FUNCTION_BLOCK FB_LICTest EXTENDS FB_TestSuite
VAR
    (* Caller-owned axis, persistent storage, and Y motor.
       In a real PRG the AxisRef would come from MAIN.Mxx. *)
    axRef    : AXIS_REF;
    fbPDS    : LCLS_Tc_DevAbs.FB_PersistentDataStorage;

    (* FB_LIC is single-axis (nActiveMotorCount := 1), so only slot 1
       holds a real motor. aiMotionStage is sized to
       MotionConstants.MAX_STATE_MOTORS to match FB_LIC.FB_Init's
       fixed-size signature; slots 2-4 default-init to a nil interface
       and are never touched. *)
    fbMotorY : FB_MotionStageNC(AxisRef := axRef, iPersistentDataStorage := fbPDS, sName := 'Y');
    aiMotionStage : ARRAY[1..MotionConstants.MAX_STATE_MOTORS] OF I_MotionStage := [fbMotorY];

    {attribute 'pytmc' := '
        pv: MMS
        astPositionState.array: 1..4
    '}
    astPositionState : ARRAY[1..MotionConstants.MAX_STATE_MOTORS]
                         OF ARRAY[1..GeneralConstants.MAX_STATES] OF ST_PositionState;

    fbFFHWO    : FB_HardwareFFOutput;
    fbArbiter  : FB_Arbiter(1);
    fbSubSysIO : FB_DummyArbIO;

    (* Per-cycle caller-owned BOOL flags passed by reference to FB_LIC. *)
    bEnableMotion         : BOOL;
    bEnableBeamParams     : BOOL;
    bEnablePositionLimits : BOOL;
    bReadDBNow            : BOOL;

    (* Device-name strings bound to FB_LIC as REFERENCE TO STRING --
       a literal cannot be REF-bound, so they live as locals here. *)
    sDeviceName    : STRING := 'TST:LIC';
    sTransitionKey : STRING := 'TST:LIC-TRANSITION';

    fbLIC : FB_LIC(
        aiMotionStage         := aiMotionStage,
        astPositionState      := astPositionState,
        fbFFHWO               := fbFFHWO,
        fbArbiter             := fbArbiter,
        sDeviceName           := sDeviceName,
        sTransitionKey        := sTransitionKey,
        bEnableMotion         := bEnableMotion,
        bEnableBeamParams     := bEnableBeamParams,
        bEnablePositionLimits := bEnablePositionLimits,
        bReadDBNow            := bReadDBNow
    );

    (* Per-install PMPS-side state config (caller-owned). Mirrors what
       a real PRG_xxL0_LIC would declare. stDefault is the caller-owned
       baseline template that FB_CC_StatePMPSConfig's inner FB_StateSetup
       preloads from; fbLIC subsequently overrides per-state sName and
       fDelta via its own FB_CC_DeviceStateDefaults array. *)
    stDefault : ST_PositionState := (
        bMoveOk       := TRUE,
        bValid        := TRUE,
        bUseRawCounts := FALSE
    );

    afbStatePMPS : ARRAY[1..4] OF FB_CC_StatePMPSConfig[
        (stPositionState := astPositionState[1][E_LIC_States.OUT],
         stDefault       := stDefault,
         fPosition       := 10,
         sPmpsState      := 'TST:LIC-OUT'),
        (stPositionState := astPositionState[1][E_LIC_States.MIRROR1],
         stDefault       := stDefault,
         fPosition       := 20,
         sPmpsState      := 'TST:LIC-MIRROR1'),
        (stPositionState := astPositionState[1][E_LIC_States.MIRROR2],
         stDefault       := stDefault,
         fPosition       := 30,
         sPmpsState      := 'TST:LIC-MIRROR2'),
        (stPositionState := astPositionState[1][E_LIC_States.TARGET],
         stDefault       := stDefault,
         fPosition       := 40,
         sPmpsState      := 'TST:LIC-TARGET')
    ];

    bFirstScan : BOOL := TRUE;
    i          : UINT;
END_VAR

(* Fake PMPS handling. *)
fbSubSysIO(
    LA  := fbArbiter,
    FFO := fbFFHWO
);

(* Caller-side PMPS configurators (per-install). *)
FOR i := 1 TO 4 DO
    afbStatePMPS[i]();
END_FOR

(* One-shot motor setup + initial caller-owned enables. Limits,
   brake/enable modes, home cmd, user/hardware enables, default
   velocity; skip NC param restore. *)
IF bFirstScan THEN
    fbMotorY.SetModeEnableLimits(
        LimBackward    := TRUE,
        LimForward     := TRUE,
        HomeEnable     := FALSE,
        BrakeMode      := E_StageBrakeMode.IF_ENABLED,
        EnableMode     := E_StageEnableMode.DURING_MOTION,
        HomeMode       := E_EpicsHomeCmd.LOW_LIMIT,
        UserEnable     := TRUE,
        HardwareEnable := TRUE
    );
    fbMotorY.SetVelocity(Velocity := 15.5);
    fbMotorY.RestoreMotionParams      := FALSE;
    fbMotorY.DoNotRestoreNcParameters := TRUE;

    bEnableMotion         := TRUE;
    bEnableBeamParams     := TRUE;
    bEnablePositionLimits := TRUE;
    bReadDBNow            := TRUE;

    bFirstScan := FALSE;
END_IF

fbPDS();
fbMotorY();
fbLIC();

TestStateMove();

METHOD TestStateMove
VAR_INST
    tonTimer   : TON;
    nIterState : UINT := 0;
END_VAR
VAR CONSTANT
    nLastState : UINT := 4; (* E_LIC_States.TARGET *)
END_VAR

(* Sanity check: can we at least move to every named state? *)
TEST('TestLICStateMove');

(* Prepare a timeout *)
tonTimer(IN := TRUE, PT := T#10s);

(* Start in Unknown, then go through the state positions one by one. *)
IF fbLIC.eEnumGet = nIterState THEN
    nIterState     := nIterState + 1;
    fbLIC.eEnumSet := nIterState;
END_IF

IF tonTimer.Q OR nIterState > nLastState THEN
    AssertFalse(tonTimer.Q, 'Timeout in LIC move test');
    TEST_FINISHED();
END_IF
END_METHOD

END_FUNCTION_BLOCK

(* stored: Version 1.1.0.1
   POU FB_LICTest: Id {ef79d59f-e709-422b-8451-9f985c309542}, SpecialFunc None
   Method TestStateMove: Id {dad8b7bd-1e01-4691-a16a-4b540b1b11f0} *)
